# EPICS autosave request: iocBoot/ioc13idd_pg3/auto_settings.req
file "spinnaker_settings.req",            P=$(P),  R=cam1:
file "NDStdArrays_settings.req",          P=$(P),  R=image1:
file "commonPlugin_settings.req",         P=$(P)
$(P)cam1:GC_BalanceWhiteAuto
$(P)cam1:GC_BlackLevel
$(P)cam1:GC_AcqFrameRateAuto
$(P)cam1:GC_GevSCPSPacketSize
